FUNCTION_BLOCK FB_EmergencyHandler EXTENDS FB_Handler
VAR_INPUT
	bReset:			BOOL;
END_VAR
VAR_OUTPUT
	bOutput:		BOOL;
END_VAR
VAR
	bResetOld: 		BOOL:= TRUE;
END_VAR

SUPER^();
IF bReset AND NOT bResetOld THEN
	bOutput:= TRUE;
END_IF
bResetOld:= bReset;

METHOD PUBLIC M_Request
VAR_INPUT
	stEvent:			ST_Event;		// event to be handled. 
END_VAR
IF stEvent.sMessage = 'Emergency Stop' THEN
	bOutput:= FALSE;
END_IF

SUPER^.M_Request(stEvent);
END_METHOD

END_FUNCTION_BLOCK

(* stored: Version 1.1.0.1, ProductVersion 3.1.4024.12
   POU FB_EmergencyHandler: Id {245b64b1-fb15-458b-96e4-a8a3c965e319}, SpecialFunc None
   Method M_Request: Id {0f74ac42-a814-4c7f-93b6-623c2e10cb5e} *)
